PROGRAM MAIN
VAR
	myReport : MyReport;
END_VAR

END_PROGRAM

(* stored: Version 1.1.0.1, ProductVersion 3.1.4024.15
   POU MAIN: Id {64f59095-be86-4f3e-8919-cb39eb9e6ff8}, SpecialFunc None *)
